FUNCTION_BLOCK TcoSequencerNonAutoRestorableTest EXTENDS TcoCore._internals_TcoContext
VAR
	_Sequencer : _TcoSequencer(THIS^, FALSE);
	_RunPLCinstanceOnce : BOOL := FALSE;
	_RunPLCinstanceCyclicaly : BOOL := FALSE;
	_StepID : INT := 32767;
	_Enabled : BOOL;
	_StepDescription : STRING := 'Last step sequence message';	
	_RunOneStep : BOOL;
	_RunAllSteps : BOOL;
	_FinishStep : BOOL;
	_Restore : BOOL;
	_CycleCount : INT;
	_RestoreCycleCount : INT;
	_Init: BOOL;
END_VAR

IF NOT _Init THEN
	ContextOpen();	
	ContextClose();	
	_Init := TRUE;
END_IF

IF _Restore THEN
	ContextOpen();	
	THIS^._Sequencer.Restore();	
	_RestoreCycleCount := _RestoreCycleCount + 1;
	_Restore := FALSE;
	ContextClose();	
	RETURN;
END_IF

IF _RunPLCinstanceOnce AND NOT _RunPLCinstanceCyclicaly THEN
	ContextOpen();	
	THIS^.PLCinstanceRun(_StepID , _Enabled, _StepDescription);
	_CycleCount := _CycleCount + 1;
	_RunPLCinstanceOnce := FALSE;
	ContextClose();	
END_IF

IF _RunPLCinstanceCyclicaly AND NOT _RunPLCinstanceOnce THEN
	ContextOpen();	
	THIS^.PLCinstanceRun(_StepID , _Enabled, _StepDescription);
	_CycleCount := _CycleCount + 1;
	ContextClose();	
END_IF

{attribute 'TcRpcEnable'}
METHOD INTERNAL ChildHasAutoRestoreEnabled : BOOL;
ChildHasAutoRestoreEnabled := _Sequencer.ChildHasAutoRestoreEnabled();
END_METHOD

{attribute 'TcRpcEnable'}
METHOD INTERNAL ChildIsAutoRestorable : BOOL;
ChildIsAutoRestorable := _Sequencer.ChildIsAutoRestorable();
END_METHOD

{attribute 'TcRpcEnable'}
METHOD INTERNAL CleanupPointers
_Sequencer.CleanupPointers();
END_METHOD

{attribute 'TcRpcEnable'}
METHOD INTERNAL ClearNumberOfSteps
_Sequencer.ClearNumberOfSteps();
END_METHOD

{attribute 'TcRpcEnable'}
METHOD INTERNAL ContextClose
SUPER^._Close();
END_METHOD

{attribute 'TcRpcEnable'}
METHOD INTERNAL ContextOpen
SUPER^._Open();
END_METHOD

{attribute 'TcRpcEnable'}
METHOD INTERNAL GetChildState : INT
GetChildState := _Sequencer.GetChildState();
END_METHOD

{attribute 'TcRpcEnable'}
METHOD INTERNAL GetCurrentStepOrder : UINT
GetCurrentStepOrder := _Sequencer._currentStep.Order;
END_METHOD

{attribute 'TcRpcEnable'}
METHOD INTERNAL GetNumberOfStepsInSequence : UINT
GetNumberOfStepsInSequence := _Sequencer._numberOfStepsInSequence;
END_METHOD

{attribute 'TcRpcEnable'}
METHOD INTERNAL GetOrderOfTheCurrentlyEvaluatedStep : UINT
GetOrderOfTheCurrentlyEvaluatedStep := _Sequencer._theOrderOfTheCurrentlyEvaluatedStep;
END_METHOD

{attribute 'TcRpcEnable'}
METHOD INTERNAL GetOrderOfTheCurrentlyExecutedStep : UINT
GetOrderOfTheCurrentlyExecutedStep := _Sequencer._theOrderOfTheCurrentlyExecutedStep;
END_METHOD

{attribute 'TcRpcEnable'}
METHOD INTERNAL GetPreviousNumberOfStepsInSequence : UINT
GetPreviousNumberOfStepsInSequence := _Sequencer._previousNumberOfStepsInSequence;
END_METHOD

{attribute 'TcRpcEnable'}
METHOD INTERNAL GetRequestStepCycle : UINT
GetRequestStepCycle := _Sequencer.RequestStepCycle;
END_METHOD

{attribute 'TcRpcEnable'}
METHOD INTERNAL GetSequencerErrorId : INT
GetSequencerErrorId := _Sequencer.GetSequencerErrorId();
END_METHOD

{attribute 'TcRpcEnable'}
METHOD INTERNAL GetTextOfTheMostImportantMessage : STRING(254)
GetTextOfTheMostImportantMessage := THIS^._Sequencer.GetTextOfTheMostImportantMessage();
END_METHOD

{attribute 'TcRpcEnable'}
METHOD INTERNAL HasAutoRestoreEnabled : BOOL;
HasAutoRestoreEnabled := _Sequencer.HasAutoRestoreEnabled();
END_METHOD

{attribute 'TcRpcEnable'}
METHOD INTERNAL IsAutoRestorable : BOOL;
IsAutoRestorable := _Sequencer.IsAutoRestorable();
END_METHOD

{attribute 'TcRpcEnable'}
METHOD INTERNAL IsFirstStepEntry : BOOL
IsFirstStepEntry := THIS^._Sequencer.IsFirstStepEntry();
END_METHOD

METHOD PROTECTED  Main
END_METHOD

{attribute 'TcRpcEnable'}
METHOD PLCinstanceRun
VAR_INPUT
	inStepId			:	UINT;
	inEnabled			:	BOOL;
	inStepDescription	:	STRING(254);	
END_VAR
THIS^._Sequencer.SetTestParams(	_RunOneStep , _RunAllSteps , _FinishStep , inStepId , inEnabled , inStepDescription);

THIS^._Sequencer.Run();
END_METHOD

{attribute 'TcRpcEnable'}
METHOD RequestStep
VAR_INPUT
	inRequestedStepId : INT;
END_VAR
_Sequencer.RequestStep(inRequestedStepId);
END_METHOD

{attribute 'TcRpcEnable'}
METHOD Restore
_Sequencer.Restore();
END_METHOD

{attribute 'TcRpcEnable'}
METHOD SequenceComplete
_Sequencer.SequenceComplete();
END_METHOD

{attribute 'TcRpcEnable'}
METHOD SequencerClose
THIS^._Sequencer.SequencerClose();
END_METHOD

{attribute 'TcRpcEnable'}
METHOD SequencerHasError : BOOL
SequencerHasError := _Sequencer.SequencerHasError();
END_METHOD

{attribute 'TcRpcEnable'}
METHOD SequencerOpen
THIS^._Sequencer.SequencerOpen();
END_METHOD

{attribute 'TcRpcEnable'}
METHOD SetChildState
VAR_INPUT
	inState			:	INT;
END_VAR
_Sequencer.SetChildState(inState);
END_METHOD

{attribute 'TcRpcEnable'}
METHOD SetCurrentStep
VAR_INPUT
	inStepID 			:	INT;
	inStepDescription	:	STRING(254);
END_VAR
_Sequencer.SetCurrentStep(inStepID := inStepID, inStepDescription := inStepDescription);
END_METHOD

{attribute 'TcRpcEnable'}
METHOD SetCyclicMode : BOOL
_Sequencer.Mode := eSequencerMode.CyclicMode;

SetCyclicMode := _Sequencer.Mode = eSequencerMode.CyclicMode;
END_METHOD

{attribute 'TcRpcEnable'}
METHOD SetNumberOfSteps : UINT
VAR_INPUT
	inNumberOfSteps :UINT;
END_VAR
_Sequencer.SetNumberOfSteps(inNumberOfSteps);
SetNumberOfSteps := _Sequencer._numberOfStepsInSequence;
END_METHOD

{attribute 'TcRpcEnable'}
METHOD SetRequestStepCycle : UINT
VAR_INPUT
	Value : UINT;
END_VAR
_Sequencer.RequestStepCycle := Value;

SetRequestStepCycle := _Sequencer.RequestStepCycle;
END_METHOD

{attribute 'TcRpcEnable'}
METHOD SetSequenceAsChecked : BOOL
VAR_INPUT
END_VAR
_Sequencer.SetSequenceAsChecked();
END_METHOD

{attribute 'TcRpcEnable'}
METHOD SetSequenceAsNotChecked : BOOL
VAR_INPUT
END_VAR
_Sequencer.SetSequenceAsNotChecked();
END_METHOD

{attribute 'TcRpcEnable'}
METHOD SetStepMode : BOOL
_Sequencer.Mode := eSequencerMode.StepMode;

SetStepMode := _Sequencer.Mode = eSequencerMode.StepMode;
END_METHOD

{attribute 'TcRpcEnable'}
METHOD Step : BOOL
VAR_INPUT
	inStepId			:	INT;
	inEnabled			:	BOOL;
	inStepDescription	:	STRING(254);		
END_VAR
Step := _Sequencer._Step(inStepID := inStepId, inEnabled := inEnabled, inStepDescription := inStepDescription);
END_METHOD

{attribute 'TcRpcEnable'}
METHOD StepBackward
_Sequencer.StepBackward();
END_METHOD

{attribute 'TcRpcEnable'}
METHOD StepCompleteWhen 
VAR_INPUT
	inCondition : BOOL;
END_VAR
_Sequencer.StepCompleteWhen(inCondition);
END_METHOD

{attribute 'TcRpcEnable'}
METHOD StepForward
_Sequencer.StepForward();
END_METHOD

{attribute 'TcRpcEnable'}
METHOD StepIn
_Sequencer.StepIn();
END_METHOD

{attribute 'TcRpcEnable'}
METHOD UpdateCurrentStepDetails
VAR_INPUT
END_VAR
_Sequencer.UpdateCurrentStepDetails();
END_METHOD

END_FUNCTION_BLOCK

(* stored: Version 1.1.0.1, ProductVersion 3.1.4024.6
   POU TcoSequencerNonAutoRestorableTest: Id {51a98037-a5c3-0526-003c-36d94696b27f}, SpecialFunc None
   Method ChildHasAutoRestoreEnabled: Id {927e7d84-c08b-0bde-39bb-9f2698695c85}
   Method ChildIsAutoRestorable: Id {95c7db10-558f-0013-0493-eedd8f38a610}
   Method CleanupPointers: Id {f261793b-5fd9-0f10-045e-c48ce347e280}
   Method ClearNumberOfSteps: Id {7bcda0f4-cc68-006d-07f7-1d794096e80e}
   Method ContextClose: Id {a2068144-8768-0cc6-2ac4-f7b57e074067}
   Method ContextOpen: Id {081c3e11-a000-09bb-3a15-0cff8a5b37be}
   Method GetChildState: Id {210b9644-e12f-03c8-3c2e-5b24f6925bb2}
   Method GetCurrentStepOrder: Id {6ad3e4e9-127e-061e-1507-35bdfe8afb19}
   Method GetNumberOfStepsInSequence: Id {d7a19c38-c019-0b93-3005-f2b003b97079}
   Method GetOrderOfTheCurrentlyEvaluatedStep: Id {4deaa7c7-014b-0c99-2264-5f70a4bb2383}
   Method GetOrderOfTheCurrentlyExecutedStep: Id {806383c1-64a4-0ae7-1d82-70ed6bd92f45}
   Method GetPreviousNumberOfStepsInSequence: Id {1491fb44-e9b5-0959-1e23-930aa0e165fc}
   Method GetRequestStepCycle: Id {f71b2f76-dfd6-06ac-1189-8dcfc7db8124}
   Method GetSequencerErrorId: Id {f13d85cd-257d-09dc-111d-e85abca68eb1}
   Method GetTextOfTheMostImportantMessage: Id {4d73dcbd-e4bb-0ae7-26b5-9400267c1c1a}
   Method HasAutoRestoreEnabled: Id {59cfae51-f09c-0054-2700-a47696981c4e}
   Method IsAutoRestorable: Id {e20dae22-b9ba-0de2-2ff3-88e481f1f9e7}
   Method IsFirstStepEntry: Id {136eb862-04d1-0ab1-33f7-59ed03a74fb3}
   Method Main: Id {29221df3-5ac3-0de8-055d-2db0206b0f5a}
   Method PLCinstanceRun: Id {b4c8497b-72b1-08fe-04a0-311bf32e037c}
   Method RequestStep: Id {07897374-03d3-0f65-3bbc-c34c3d9b721c}
   Method Restore: Id {ed039be1-5ec9-0f31-1ced-279adddd1155}
   Method SequenceComplete: Id {99caabcc-a19b-0b51-39fd-9a25f213e16d}
   Method SequencerClose: Id {f7829c9b-5f03-09e8-0641-8171778ff555}
   Method SequencerHasError: Id {9e1664b3-73ed-07a4-2a34-a272c5fff16f}
   Method SequencerOpen: Id {d1b26862-be46-0bba-2e13-0ed45cf8aa9a}
   Method SetChildState: Id {5763788a-36fa-0e64-0317-b960304583c2}
   Method SetCurrentStep: Id {aae831a2-eb4c-0fda-2f20-425fc5ae0b6c}
   Method SetCyclicMode: Id {81ab4539-ac96-04ea-1033-d164e828e90d}
   Method SetNumberOfSteps: Id {8f816cfa-b5d2-0b69-35c7-36d1b3cf0fa8}
   Method SetRequestStepCycle: Id {ec311bd2-8210-0230-37a9-db99310da642}
   Method SetSequenceAsChecked: Id {5533a50f-9c90-0fcf-1640-6737f926030a}
   Method SetSequenceAsNotChecked: Id {a96b87cc-33c0-0351-3dbf-db3ac932ab2f}
   Method SetStepMode: Id {ce8881b6-9e87-058a-23ac-981a9ce728d8}
   Method Step: Id {9a4fa3e9-79a9-0600-1f4e-25000370363d}
   Method StepBackward: Id {d98107a1-3a0d-0df5-09e6-118646b66a3a}
   Method StepCompleteWhen: Id {528973e4-bd1c-0a49-38fe-907c102d8f6a}
   Method StepForward: Id {8497da56-753d-0a4d-1dbe-11b2662ecbb5}
   Method StepIn: Id {f134033d-36eb-0445-25df-ab96ab833503}
   Method UpdateCurrentStepDetails: Id {44a4b22c-60d5-0113-140a-edda3c2eedd4} *)
